{attribute addProperty BoxType "EPP6228-0022-0016"}
{attribute addProperty Id "Pin2_Ch1AT %I*BOOL811Pin2_Ch2AT %I*BOOL812Pin2_Ch3AT %I*BOOL813Pin2_Ch4AT %I*BOOL814Pin2_Ch5AT %I*BOOL815Pin2_Ch6AT %I*BOOL816Pin2_Ch7AT %I*BOOL817Pin2_Ch8AT %I*BOOL818"}
{attribute addProperty CRC "3528142583"}
{attribute addProperty SizeInBites "64"}
{attribute addProperty SizeInBytes "8"}
TYPE Digital_Inputs_D24B2EF7 :
STRUCT
	{attribute addProperty Name "Pin2_Ch1"}
	Pin2_Ch1 AT %I* : BOOL;
	{attribute addProperty Name "Pin2_Ch2"}
	Pin2_Ch2 AT %I* : BOOL;
	{attribute addProperty Name "Pin2_Ch3"}
	Pin2_Ch3 AT %I* : BOOL;
	{attribute addProperty Name "Pin2_Ch4"}
	Pin2_Ch4 AT %I* : BOOL;
	{attribute addProperty Name "Pin2_Ch5"}
	Pin2_Ch5 AT %I* : BOOL;
	{attribute addProperty Name "Pin2_Ch6"}
	Pin2_Ch6 AT %I* : BOOL;
	{attribute addProperty Name "Pin2_Ch7"}
	Pin2_Ch7 AT %I* : BOOL;
	{attribute addProperty Name "Pin2_Ch8"}
	Pin2_Ch8 AT %I* : BOOL;
END_STRUCT
END_TYPE

(* stored: Version 1.2.0.0, ProductVersion 3.1.4024.9
   DUT Digital_Inputs_D24B2EF7: Id {99dcaf0d-77f8-479d-8e38-52586bbd9f1d} *)
